// TIA Portal project "S7netTiaProject(WaterLevelControl_discrete)" (V16)

(* hardware
DEVICE "S7-1200 station_1"  S7-1200 Station
   slot 0: "Rack_0"  S7-1200 Rack  Rack  V1.0
   slot 1: "PLC_1"  CPU 1214C DC/DC/DC  6ES7 214-1AG40-0XB0  V4.4
DEVICE "HMI_1"  KTP900 Basic PN
   slot 0: "HMI_1"  KTP900 Basic PN  6AV2 123-2JB03-0AX0  16.0.0.0
   slot 1: "HMI_RT_1"  KTP900 Basic PN  6AV2 123-2JB03-0AX0  16.0.0.0
   slot 5: "HMI_1.IE_CP_1"  PROFINET Interface  16.0.0.0
      slot 1: "PROFINET Interface_1"  PROFINET Interface
         slot 1: "Port_1"  Port
*)

// ===== PLC "PLC_1"  CPU 1214C DC/DC/DC =====

VAR_GLOBAL   // PLC tag table "Default tag table"
   "start" AT %M0.0 : Bool;
   "Motor" AT %M0.1 : Bool;
   "S1_memory" AT %M0.2 : Bool;
   "S2_memory" AT %M0.3 : Bool;
   "S3_val" AT %MD2 : Real;
   "level" AT %MD6 : Real;
END_VAR

DATA_BLOCK "DataBlock1"   // DB1
{ S7_Optimized_Access := 'FALSE' }
VERSION : 0.1
   VAR
      S1 : Bool := false;
      S2 : Bool;
      S3 : Int;
      M1 : Int;
      K1 : Int;
      Start : Bool := false;
      Stop : Bool;
   END_VAR
BEGIN
END_DATA_BLOCK

ORGANIZATION_BLOCK "Main"   // OB1, LAD, ProgramCycle
TITLE = "Main Program Sweep (Cycle)"
{ S7_Optimized_Access := 'TRUE' }
VERSION : 0.1
   VAR_INPUT
      Initial_Call : Bool;   // Initial call of this OB
      Remanence : Bool;   // =True, if remanent data are available
   END_VAR
BEGIN

REGION Network 1
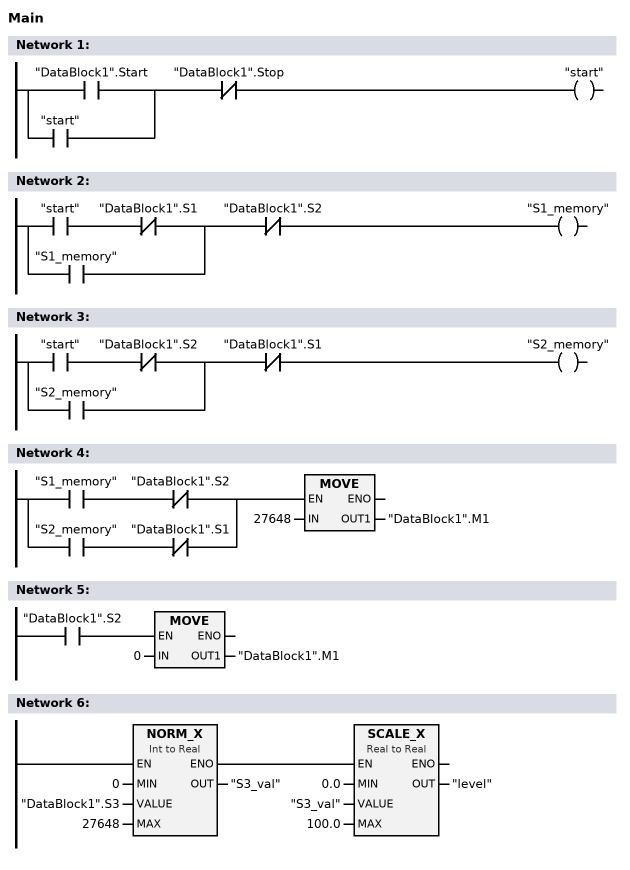
   RUNG wire#powerrail
      Contact( "DataBlock1".Start )
      wire#w1
      I_Contact( "DataBlock1".Stop )
      Coil( "start" )
   END_RUNG
   RUNG wire#powerrail
      Contact( "start" )
   END_RUNG wire#w1
   // the same network as SCL:
   "start" := ("DataBlock1".Start OR "start") AND NOT "DataBlock1".Stop;
END_REGION

REGION Network 2
   RUNG wire#powerrail
      Contact( "start" )
      I_Contact( "DataBlock1".S1 )
      wire#w1
      I_Contact( "DataBlock1".S2 )
      Coil( "S1_memory" )
   END_RUNG
   RUNG wire#powerrail
      Contact( "S1_memory" )
   END_RUNG wire#w1
   // the same network as SCL:
   "S1_memory" := (("start" AND NOT "DataBlock1".S1) OR "S1_memory") AND NOT "DataBlock1".S2;
END_REGION

REGION Network 3
   RUNG wire#powerrail
      Contact( "start" )
      I_Contact( "DataBlock1".S2 )
      wire#w1
      I_Contact( "DataBlock1".S1 )
      Coil( "S2_memory" )
   END_RUNG
   RUNG wire#powerrail
      Contact( "S2_memory" )
   END_RUNG wire#w1
   // the same network as SCL:
   "S2_memory" := (("start" AND NOT "DataBlock1".S2) OR "S2_memory") AND NOT "DataBlock1".S1;
END_REGION

REGION Network 4
   RUNG wire#powerrail
      Contact( "S1_memory" )
      I_Contact( "DataBlock1".S2 )
      wire#w1
      Move(in := 27648, out1 => "DataBlock1".M1)
   END_RUNG
   RUNG wire#powerrail
      Contact( "S2_memory" )
      I_Contact( "DataBlock1".S1 )
   END_RUNG wire#w1
   // the same network as SCL:
   IF ("S1_memory" AND NOT "DataBlock1".S2) OR ("S2_memory" AND NOT "DataBlock1".S1) THEN
       "DataBlock1".M1 := 27648;
   END_IF;
END_REGION

REGION Network 5
   RUNG wire#powerrail
      Contact( "DataBlock1".S2 )
      Move(in := 0, out1 => "DataBlock1".M1)
   END_RUNG
   // the same network as SCL:
   IF "DataBlock1".S2 THEN "DataBlock1".M1 := 0; END_IF;
END_REGION

REGION Network 6
   RUNG wire#powerrail
      { S7_Templates := "[SrcType := Int, DestType := Real]" } Normalize(min := 0, value := "DataBlock1".S3, max := 27648, out => "S3_val")
      { S7_Templates := "[SrcType := Real, DestType := Real]" } Scale(min := 0.0, value := "S3_val", max := 100.0, out => "level")
   END_RUNG
   // the same network as SCL:
   "S3_val" := NORM_X(MIN := 0, VALUE := "DataBlock1".S3, MAX := 27648);
   "level" := SCALE_X(MIN := 0.0, VALUE := "S3_val", MAX := 100.0);
END_REGION
END_ORGANIZATION_BLOCK

(* ===== HMI "HMI_RT_1" =====
system functions are stored by id; their names below are inferred from use
connection "HMI_Connection_1": ETHERNET, SMART_S7_1200_OMS

HMI tags "Default tag table"
   "Tag_ScreenNumber" : UInt, internal
   "level" : Real = PLC level AT %MD6, 1 s
   "DataBlock1_Start" : Bool = PLC DataBlock1.Start AT %DB1.DBX8.0, 1 s
   "DataBlock1_Stop" : Bool = PLC DataBlock1.Stop AT %DB1.DBX8.1, 1 s

Template "Template_1" 800x480
   Button "Exit" at 722,440 size 55x39; TextOff 'Exit'; PictureOff "ExitRuntime_KTP900_Basic_PN_TR"; PictureOn "ExitRuntime_KTP900_Basic_PN_TR"
      on Release: StopRuntime(0)
   Button "Template_Button" at 622,440 size 55x39; TextOff 'Text'
   Button "Template_Button_1" at 522,440 size 55x39; TextOff 'Text'
   Button "Template_Button_2" at 422,440 size 55x39; TextOff 'Text'
   Button "Template_Button_3" at 322,440 size 55x39; TextOff 'Text'
   Button "Template_Button_4" at 222,440 size 55x39; TextOff 'Text'
   Button "Alarms" at 122,440 size 55x39; TextOff 'Alarms'; PictureOff "AlarmDisplay_KTP900_Basic_PN_TR"; PictureOn "AlarmDisplay_KTP900_Basic_PN_TR"
      on Release: function_ef3f5d25("Alarm window_Unacknowledged", -1)
   Button "Start screen" at 22,440 size 55x39; TextOff 'Start screen'; PictureOff "NavigateHome_KTP900_Basic_PN_TR"; PictureOn "NavigateHome_KTP900_Basic_PN_TR"
      on Release: ActivateScreen("Root screen", 0)
   SymbolicIOField "Symbolic_IO_Field_Screen" at 73,7 size 620x26; TextOff '0'; TextOn '1'; TextList "TextList_ScreenNames"
      ProcessValue <- "Tag_ScreenNumber"
      on Change: ActivateScreenByNumber("Tag_ScreenNumber", 0)
   DateTimeField "HmiScreenItemData" at 695,20 size 105x20
   DateTimeField "HmiScreenItemData_1" at 695,0 size 105x20
   GraphicView "Logo" at 0,0 size 71x40; Picture "Logo of HMI_1"

screen "Root screen" 800x480, template "Template_1"
   on GenerateScreen: SetTag("Tag_ScreenNumber", 1)
   TextField "HmiScreenItemData" at 80,226 size 640x22; Text 'Welcome to HMI_1 (KTP900 Basic+ PN)!'

screen "Screen_1" 800x480
   Button "Button_1" at 23,19 size 96x32; TextOff 'Start'
      on Press: SetBit("DataBlock1_Start")
      on Release: ResetBit("DataBlock1_Start")
   Button "Button_2" at 144,19 size 96x32; TextOff 'Stop'
      on Press: SetBit("DataBlock1_Stop")
      on Release: ResetBit("DataBlock1_Stop")
   TrendView "Trend view_2" at 99,107 size 600x300
*)